// TwinCAT 3 PLC project Untitled1
// ProgramVersion: 3.1.4023.0
// libraries:
//   Tc2_Standard, * (Beckhoff Automation GmbH)
//   Tc2_System, * (Beckhoff Automation GmbH)
//   Tc3_Module, * (Beckhoff Automation GmbH)
// project tree:
//   / PlcTask.TcTTO
//   POUs/ MAIN.TcPOU
// real-time tasks:
//   TASK PlcTask: cycle T#10ms, priority 20, ADS port 350
// I/O:
//   DEVICE Device 1 (EtherCAT), AmsNetId 5.131.216.41.2.1
//     Term 1 (EK1200) [EK1200-5000 EtherCAT Power supply (2A E-Bus)]
//       Term 2 (EL2809) [EL2809 16Ch. Dig. Output 24V, 0.5A]
//       Term 3 (EL6695) [EL6695 EtherCAT Bridge terminal (Primary)]
//       Term 4 (EK1122) [EK1122 2 port EtherCAT junction]
//         Term 5 (EK1100) [EK1100 EtherCAT Coupler (2A E-Bus)]
//           Term 6 (EL1809) [EL1809 16Ch. Dig. Input 24V, 3ms]
//           Term 7 (EL2809) [EL2809 16Ch. Dig. Output 24V, 0.5A]
//           Term 8 (EL9011) [EL9011 End Terminal]
// variable links:
//   Untitled1/Untitled1 Instance <-> Device 1 (EtherCAT)/Term 1 (EK1200)/Term 4 (EK1122)/Term 5 (EK1100)/Term 6 (EL1809)
//     PlcTask Inputs/MAIN.done <-> Channel 4/Input
//     PlcTask Inputs/MAIN.error <-> Channel 1/Input
//     PlcTask Inputs/MAIN.home <-> Channel 5/Input
//     PlcTask Inputs/MAIN.ready <-> Channel 2/Input
//   Untitled1/Untitled1 Instance <-> Device 1 (EtherCAT)/Term 1 (EK1200)/Term 4 (EK1122)/Term 5 (EK1100)/Term 7 (EL2809)
//     PlcTask Outputs/MAIN.enable <-> Channel 2/Output
//     PlcTask Outputs/MAIN.execute <-> Channel 1/Output
//     PlcTask Outputs/MAIN.reset <-> Channel 3/Output

CONFIGURATION Untitled1
    RESOURCE PLC ON TwinCAT3
        TASK PlcTask(INTERVAL := T#10ms, PRIORITY := 20);
        PROGRAM MAIN WITH PlcTask : MAIN;
    END_RESOURCE
END_CONFIGURATION

// ---- POUs/MAIN.TcPOU
PROGRAM MAIN
VAR
	manual : BOOL; //:= TRUE;
	
	error AT %I* : BOOL;
	ready AT %I* : BOOL;
	//busy AT %I* : BOOL;
	done AT %I* : BOOL;
	home AT %I* : BOOL;
	
	execute AT %Q* : BOOL;
	enable AT %Q* : BOOL;
	reset AT %Q* : BOOL;

	start : BOOL;
	
	timeout : TON;
	hold : TON;
	
	step : (SETUP, STRAP, WAIT);
	
	i : INT;
END_VAR
VAR CONSTANT
	pulseWidth : TIME := T#500MS;
	delayTime : TIME := T#500MS;
	
	failTime : TIME := T#30S;
END_VAR

hold(IN:= , PT:= delayTime, Q=> , ET=> );
timeout(IN:= step > SETUP, PT:= failTime, Q=> , ET=> );

IF timeout.Q THEN
	timeout.IN := FALSE;
	step := SETUP;
END_IF

IF manual THEN
	RETURN;
END_IF

CASE step OF	
	SETUP:
		//reset := NOT reset;
		//enable := NOT enable;
		
		IF NOT error THEN
			reset := FALSE;
			enable := TRUE;
			
			IF start THEN
				start := FALSE;
				step := STRAP;
			END_IF
			
		ELSE
			reset := NOT reset;
			enable := NOT enable;
		END_IF
	
	STRAP:
		IF NOT execute THEN
			execute := TRUE;
			RETURN;
		END_IF
		
		IF execute AND NOT home THEN
			execute := FALSE;
			step := WAIT;
		END_IF
		
	WAIT:
		IF home THEN
			hold.IN := TRUE;
			enable := FALSE;
			execute := FALSE;
		END_IF
		
		IF hold.Q THEN
			hold.IN := FALSE;
			i := i + 1;
			step := 0;			
		END_IF
END_CASE

END_PROGRAM
